// TIA Portal V18 export
DATA_BLOCK "fbProcessControlSCL_DB"   // DB2
// stored: InstanceOfName fbProcessControlSCL, InstanceOfType FB
"fbProcessControlSCL"
   // VAR_INPUT
   //    iTemperature : Int;
   //    iTarget : Int;
   // END_VAR
   // VAR_OUTPUT
   //    oTemperatureTooHigh : Bool;
   //    oTemperatureTooLow : Bool;
   // END_VAR
   // VAR_IN_OUT
   //    InOut_1 : Bool;
   // END_VAR
BEGIN
END_DATA_BLOCK
